SUBAPPLICATION AX_GT_0_UINT (* Prüft ob UINT-Adapter Wert > 0 ist (AX-Adapter Ausgang) *)
  (* Standard: 61499-2 *)
  (* Version 1.0, 2026-04-20, franz *)
  PACKAGE MyLib::sys;
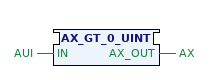
  SOCKETS
    IN : adapter::types::unidirectional::AUI;
  END_SOCKETS
  PLUGS
    AX_OUT : adapter::types::unidirectional::AX;
  END_PLUGS
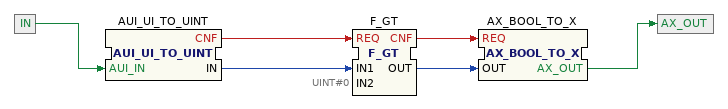
  FBS
    AUI_UI_TO_UINT : adapter::conversion::unidirectional::AUI_UI_TO_UINT;
    AX_BOOL_TO_X : adapter::conversion::unidirectional::AX_BOOL_TO_X;
    F_GT : iec61131::comparison::F_GT(IN2 := UINT#0);
  END_FBS
  EVENT_CONNECTIONS
    AUI_UI_TO_UINT.CNF TO F_GT.REQ;
    F_GT.CNF TO AX_BOOL_TO_X.REQ;
  END_CONNECTIONS
  DATA_CONNECTIONS
    AUI_UI_TO_UINT.IN TO F_GT.IN1;
    F_GT.OUT TO AX_BOOL_TO_X.OUT;
  END_CONNECTIONS
  ADAPTER_CONNECTIONS
    IN TO AUI_UI_TO_UINT.AUI_IN;
    AX_BOOL_TO_X.AX_OUT TO AX_OUT;
  END_CONNECTIONS
END_SUBAPPLICATION
